(* IEC 61131-3 sources: TSA-FMICS22/ahorn/test/benchmark/dissertation/SA, 2 files *)

(* ---- FlattenedSFAntivalent.st ---- *)
PROGRAM SFAntivalent
VAR_INPUT
    Activate : BOOL;
    SChannelNC : SAFEBOOL;
    SChannelNO : SAFEBOOL;
    DiscrepancyTime : TIME;
END_VAR
VAR
    Timer : TON;
    TimerQ : BOOL;
    TimerET : TIME;
END_VAR
VAR_OUTPUT
    Ready : BOOL;
    SAntivalentOut : BOOL;
    Error : BOOL;
    DiagCode : WORD;
END_VAR

IF NOT Activate THEN
    DiagCode := 16#0000;
ELSE
    CASE DiagCode OF
    16#0000:
        IF Activate THEN
            DiagCode := 16#8001;
        END_IF;
    16#8001:
        IF SChannelNC AND SChannelNO THEN
            DiagCode := 16#8004;
            Timer(IN:=TRUE, PT:=DiscrepancyTime, Q=>TimerQ, ET=>TimerET);
        ELSIF NOT SChannelNC AND NOT SChannelNO THEN
            DiagCode := 16#8014;
            Timer(IN:=TRUE, PT:=DiscrepancyTime, Q=>TimerQ, ET=>TimerET);
        ELSIF SChannelNC AND NOT SChannelNO THEN
            DiagCode := 16#8000;
        END_IF;
    16#8004:
        IF TimerQ THEN
            DiagCode := 16#C001;
        ELSIF NOT SChannelNC THEN
            DiagCode := 16#8001;
        ELSIF NOT SChannelNO THEN
            DiagCode := 16#8000;
        END_IF;
    16#C001,
    16#C002:
        IF NOT SChannelNC AND SChannelNO THEN
            DiagCode := 16#8001;
        END_IF;
    16#8014:
        IF TimerQ THEN
            DiagCode := 16#C002;
        ELSIF SChannelNO THEN
            DiagCode := 16#8001;
        ELSIF SChannelNC THEN
            DiagCode := 16#8000;
        END_IF;
    16#C003:
        IF NOT SChannelNC AND SChannelNO THEN
            DiagCode := 16#8001;
        END_IF;
    16#8005:
        IF TimerQ THEN
            DiagCode := 16#C003;
        ELSIF NOT SChannelNC AND SChannelNO THEN
            DiagCode := 16#8001;
        END_IF;
    16#8000:
        IF NOT SChannelNC OR SChannelNO THEN
            DiagCode := 16#8005;
            Timer(IN:=TRUE, PT:=DiscrepancyTime, Q=>TimerQ, ET=>TimerET);
        ELSIF NOT SChannelNC AND SChannelNO THEN
            DiagCode := 16#8001;
        END_IF;
    END_CASE;
END_IF;

CASE DiagCode OF
16#0000:
    Timer(IN:=FALSE, PT:=DiscrepancyTime, Q=>TimerQ, ET=>TimerET);
    Ready := FALSE;
    Error := FALSE;
    SAntivalentOut:= FALSE;
16#8000:
    Timer(IN:=FALSE, PT:=DiscrepancyTime, Q=>TimerQ, ET=>TimerET);
    Ready := TRUE;
    Error := FALSE;
    SAntivalentOut := TRUE;
16#8001:
    Timer(IN:=FALSE, PT:=DiscrepancyTime, Q=>TimerQ, ET=>TimerET);
    Ready := TRUE;
    Error := FALSE;
    SAntivalentOut:= FALSE;
16#8004,
16#8014,
16#8005:
    Timer(IN:=TRUE, PT:=DiscrepancyTime, Q=>TimerQ, ET=>TimerET);
    Ready := TRUE;
    Error := FALSE;
    SAntivalentOut:= FALSE;
16#C001,
16#C002,
16#C003:
    Timer(IN:=FALSE, PT:=DiscrepancyTime, Q=>TimerQ, ET=>TimerET);
    Ready := TRUE;
    Error := TRUE;
    SAntivalentOut:= FALSE;
END_CASE;
END_PROGRAM

FUNCTION_BLOCK TON
VAR_INPUT
    IN : BOOL;
    PT : TIME;
END_VAR
VAR
    running : BOOL;
END_VAR
VAR_TEMP
    timeout : BOOL;
END_VAR
VAR_OUTPUT
    Q : BOOL;
    ET : TIME;
END_VAR
timeout := NONDETERMINISTIC_BOOL();
IF NOT IN THEN
    Q := FALSE;
    running := FALSE;
ELSIF NOT running AND NOT Q THEN
    running := TRUE;
ELSIF running AND NOT Q THEN
    Q := timeout;
    running := NOT Q;
END_IF;
ET := NONDETERMINISTIC_TIME();
END_FUNCTION_BLOCK

(* ---- FlattenedSFEDM.st ---- *)
PROGRAM SFEDM
VAR_INPUT
    Activate : BOOL ;
    SOutControl	: SAFEBOOL ;
    SEDM1 : SAFEBOOL ;
    SEDM2 : SAFEBOOL ;
    MonitoringTime : TIME;
    SStartReset	: SAFEBOOL ;
    Reset : BOOL ;
END_VAR
VAR
    Timer : TON;
    TimerQ : BOOL;
    TimerET : TIME;
    RTRIGatReset : RTRIG;
    RTRIGatResetQ : BOOL;
    RTRIGatOutControl : RTRIG;
    RTRIGatOutControlQ : BOOL;
    RTRIGatEDM1 : RTRIG;
    RTRIGatEDM1Q : BOOL;
    RTRIGatEDM2	: RTRIG;
    RTRIGatEDM2Q : BOOL;
END_VAR
VAR_OUTPUT
    Ready : BOOL ;
    SEDMOut	: SAFEBOOL ;
    Error : BOOL ;
    DiagCode : WORD:=16#0000 ;
END_VAR
(* Rising edge detection *)
RTRIGatReset(CLK:=Reset, Q=>RTRIGatResetQ);
RTRIGatOutControl(CLK:=SOutControl, Q=>RTRIGatOutControlQ);
RTRIGatEDM1(CLK:=SEDM1, Q=>RTRIGatEDM1Q);
RTRIGatEDM2(CLK:=SEDM2, Q=>RTRIGatEDM2Q);
IF NOT Activate THEN
    DiagCode := 16#0000;
ELSE
    CASE DiagCode OF
    16#0000:
        IF Activate THEN
            DiagCode := 16#8001;
        END_IF;
    16#8000:
        IF TimerQ AND SEDM1 AND NOT SEDM2 THEN
            DiagCode := 16#C070;
        ELSIF TimerQ AND NOT SEDM1 AND SEDM2 THEN
            DiagCode := 16#C080;
        ELSIF TimerQ AND SEDM1 AND SEDM2 THEN
            DiagCode := 16#C090;
        ELSIF NOT SOutControl THEN
            DiagCode := 16#8010;
            Timer(IN:=FALSE, PT:=MonitoringTime, Q=>TimerQ, ET=>TimerET);
        END_IF;
    16#8001:
        IF Reset AND NOT RTRIGatResetQ AND NOT SStartReset THEN
            DiagCode := 16#C001;
        ELSIF RTRIGatResetQ AND RTRIGatOutControlQ AND NOT SStartReset THEN
            DiagCode := 16#C111;
        ELSIF RTRIGatResetQ OR SStartReset THEN
            DiagCode := 16#8010;
            Timer(IN:=FALSE, PT:=MonitoringTime, Q=>TimerQ, ET=>TimerET);
        END_IF;
    16#8010:
        IF SOutControl AND NOT SEDM1 AND SEDM2 THEN
            DiagCode := 16#C010;
        ELSIF SOutControl AND SEDM1 AND NOT SEDM2 THEN
            DiagCode := 16#C020;
        ELSIF SOutControl AND NOT SEDM1 AND NOT SEDM2 THEN
            DiagCode := 16#C030;
        ELSIF TimerQ AND NOT SEDM1 AND SEDM2 THEN
            DiagCode := 16#C040;
        ELSIF TimerQ AND SEDM1 AND NOT SEDM2 THEN
            DiagCode := 16#C050;
        ELSIF TimerQ AND NOT SEDM1 AND NOT SEDM2 THEN
            DiagCode := 16#C060;
        ELSIF SOutControl THEN
            DiagCode := 16#8000;
            Timer(IN:=FALSE, PT:=MonitoringTime, Q=>TimerQ, ET=>TimerET);
        END_IF;
    16#C001:
        IF NOT Reset THEN
            DiagCode := 16#8001;
        END_IF;
    16#C010, 16#C020, 16#C030:
        IF (Reset AND NOT RTRIGatResetQ AND SEDM1 AND SEDM2) OR (RTRIGatResetQ AND RTRIGatEDM1Q AND NOT RTRIGatEDM2Q) THEN
            DiagCode := 16#C011;
        ELSIF (Reset AND NOT RTRIGatResetQ AND SEDM1 AND SEDM2) OR (RTRIGatResetQ AND NOT RTRIGatEDM1Q AND RTRIGatEDM2Q) THEN
            DiagCode := 16#C021;
        ELSIF (Reset AND NOT RTRIGatResetQ AND SEDM1 AND SEDM2) OR (RTRIGatResetQ AND RTRIGatEDM1Q AND RTRIGatEDM2Q) THEN
            DiagCode := 16#C031;
        ELSIF RTRIGatResetQ AND SEDM1 AND SEDM2 THEN
            DiagCode := 16#8010;
            Timer(IN:=FALSE, PT:=MonitoringTime, Q=>TimerQ, ET=>TimerET);
        END_IF;
    16#C011:
        IF NOT Reset THEN
            DiagCode := 16#C010;
        END_IF;
    16#C021:
        IF NOT Reset THEN
            DiagCode := 16#C020;
        END_IF;
    16#C031:
        IF NOT Reset THEN
            DiagCode := 16#C030;
        END_IF;
    16#C040, 16#C050, 16#C060:
        IF (Reset AND NOT RTRIGatResetQ AND SEDM1 AND SEDM2) OR (RTRIGatResetQ AND RTRIGatEDM1Q AND NOT RTRIGatEDM2Q) THEN
            DiagCode := 16#C041;
        ELSIF (Reset AND NOT RTRIGatResetQ AND SEDM1 AND SEDM2) OR (RTRIGatResetQ AND NOT RTRIGatEDM1Q AND RTRIGatEDM2Q) THEN
            DiagCode := 16#C051;
        ELSIF (Reset AND NOT RTRIGatResetQ AND SEDM1 AND SEDM2) OR (RTRIGatResetQ AND RTRIGatEDM1Q AND RTRIGatEDM2Q) THEN
            DiagCode := 16#C061;
        ELSIF RTRIGatResetQ AND SEDM1 AND SEDM2 THEN
            DiagCode := 16#8010;
            Timer(IN:=FALSE, PT:=MonitoringTime, Q=>TimerQ, ET=>TimerET);
        END_IF;
    16#C041:
        IF NOT Reset THEN
            DiagCode := 16#C040;
        END_IF;
    16#C051:
        IF NOT Reset THEN
            DiagCode := 16#C050;
        END_IF;
    16#C061:
        IF NOT Reset THEN
            DiagCode := 16#C060;
        END_IF;
    16#C070:
        IF Reset AND NOT RTRIGatResetQ THEN
            DiagCode := 16#C071;
        ELSIF RTRIGatResetQ AND NOT (RTRIGatEDM1Q OR RTRIGatEDM2Q) THEN
            DiagCode := 16#8010;
            Timer(IN:=FALSE, PT:=MonitoringTime, Q=>TimerQ, ET=>TimerET);
        END_IF;
    16#C080:
        IF Reset AND NOT RTRIGatResetQ THEN
            DiagCode := 16#C081;
        ELSIF RTRIGatResetQ AND NOT (RTRIGatEDM1Q OR RTRIGatEDM2Q) THEN
            DiagCode := 16#8010;
            Timer(IN:=FALSE, PT:=MonitoringTime, Q=>TimerQ, ET=>TimerET);
        END_IF;
    16#C090:
        IF Reset AND NOT RTRIGatResetQ THEN
            DiagCode := 16#C091;
        ELSIF RTRIGatResetQ AND NOT (RTRIGatEDM1Q OR RTRIGatEDM2Q) THEN
            DiagCode := 16#8010;
            Timer(IN:=FALSE, PT:=MonitoringTime, Q=>TimerQ, ET=>TimerET);
        END_IF;
    16#C071:
        IF NOT Reset THEN
            DiagCode := 16#C070;
        END_IF;
    16#C081:
        IF NOT Reset THEN
            DiagCode := 16#C080;
        END_IF;
    16#C091:
        IF NOT Reset THEN
            DiagCode := 16#C090;
        END_IF;
    16#C111:
        IF NOT Reset THEN
            DiagCode := 16#8001;
        END_IF;
    END_CASE;
END_IF;
CASE DiagCode OF
16#0000:
    Ready := FALSE;
    SEDMOut := FALSE;
    Error := FALSE;
16#8001:
    Ready := TRUE;
    SEDMOut := FALSE;
    Error := FALSE;
16#8010:
    Ready := TRUE;
    SEDMOut := FALSE;
    Error := FALSE;
    Timer(IN:=TRUE, PT:=MonitoringTime, Q=>TimerQ, ET=>TimerET);
16#8000:
    Ready := TRUE;
    SEDMOut := TRUE;
    Error := FALSE;
    Timer(IN:=TRUE, PT:=MonitoringTime, Q=>TimerQ, ET=>TimerET);
16#C001, 16#C010, 16#C011, 16#C020, 16#C021, 16#C030, 16#C031, 16#C040, 16#C041, 16#C050, 16#C051, 16#C060, 16#C061, 16#C070, 16#C071, 16#C080, 16#C081, 16#C090, 16#C091, 16#C111:
    Ready := TRUE;
    SEDMOut := FALSE;
    Error := TRUE;
END_CASE;
END_PROGRAM

FUNCTION_BLOCK TON
VAR_INPUT
    IN : BOOL;
    PT : TIME;
END_VAR
VAR
    running : BOOL;
END_VAR
VAR_TEMP
    timeout : BOOL;
END_VAR
VAR_OUTPUT
    Q : BOOL;
    ET : TIME;
END_VAR
timeout := NONDETERMINISTIC_BOOL();
IF NOT IN THEN
    Q := FALSE;
    running := FALSE;
ELSIF NOT running AND NOT Q THEN
    running := TRUE;
ELSIF running AND NOT Q THEN
    Q := timeout;
    running := NOT Q;
END_IF;
ET := NONDETERMINISTIC_TIME();
END_FUNCTION_BLOCK

FUNCTION_BLOCK RTRIG
VAR_INPUT
    CLK : BOOL;
END_VAR
VAR
    M : BOOL;
END_VAR
VAR_OUTPUT
    Q : BOOL;
END_VAR
    Q := CLK AND NOT M;
    M := CLK;
END_FUNCTION_BLOCK
